(* PLC project CoDeSys External Library Template, WAGO e!COCKPIT e!COCKPIT, author 3S - Smart Software Solutions GmbH *)
(* stored: creationDateTime 2019-10-29T12:22:40.9809376, version 3.5.5.30, modificationDateTime 2019-10-24T14:40:07.960949, organization 3S - Smart Software Solutions GmbH *)
(* Library project template with all possible element types, docu and a sample project structure *)

FUNCTION fnTablicaKomunikatowInkrementacja : BOOL
  VAR_INPUT
    intRozmiarTablicy : INT;
  END_VAR
  VAR_IN_OUT
    intWskaznik : INT;
  END_VAR

            intWskaznik := 	intWskaznik + 1; 
IF intWskaznik > intRozmiarTablicy THEN
	intWskaznik := 1;
END_IF

          
END_FUNCTION
